(*********************************** G.D S.p.A. - Technical Department ***********************************
============= PROGRAM INFO ============
FOLDER:             TBD
MACHINES INVOLVED:  TBD 

============= DESCRIPTION =============
csp machine declaration

============= REVISIONS ===============
Date		Version	 	Author      	Description             
----------	-------		------------  	--------------------------------------------
2020/02/19 	0000.00	 	G.Imbriaco		

**********************************************************************************************************)
(*$R process_ref := prc; $*)
PROGRAM csp_case_glue_os_guns
VAR
	
	prc:											process;
	prc_path:										STRING;
	
END_VAR

VAR CONSTANT

END_VAR

_read_var_input();
_read_var_input();

_object_manager();

IF 	NOT objects_running()
THEN
	RETURN;	
END_IF

_read_process_image();

_mode_manager();

CASE process_get_mode(prc) of
	MODE_ABSENT,
	MODE_INACTIVE:
		RETURN;
	MODE_TEST:
		_handle_process_test();
END_CASE

_set_runtime_properties();

(********************************* BODY *********************************)

(************************************************************************)

_handle_messages();

_write_output();

ACTION _handle_messages:
;
END_ACTION

ACTION _handle_process_test:
;
END_ACTION

ACTION _mode_manager:
IF process_mode_req_is_pending(prc)
THEN
    process_apply_mode_req_first_step(prc);
    CASE process_get_mode(prc) OF
        MODE_TO_ABSENT:
			;
        MODE_TO_INACTIVE:
			;
        MODE_TO_TEST:
			;
        MODE_TO_OPERATIONAL:
			;
    END_CASE
    process_apply_mode_req_second_step(prc);
END_IF
END_ACTION

ACTION _object_manager:
IF objects_initialization()
THEN
	sub_process_init(
		object_name					:= 'csp_case_glue_os_guns.prc', 
		process						:= csp_case_glue_os.prc, 
		CONVERSION_this				:= prc);
		
	prc_path 						:= process_get_path(prc);
	
END_IF

IF objects_running()
THEN
	process_cycle(prc);

END_IF
END_ACTION

ACTION _read_process_image:
;
END_ACTION

ACTION _read_var_input:
;
END_ACTION

ACTION _set_runtime_properties:
;
END_ACTION

ACTION _write_output:
;
END_ACTION

END_PROGRAM

(* stored: Version 1.1.0.1, ProductVersion 3.1.4024.3
   POU csp_case_glue_os_guns: Id {7930b6d0-f08d-41ac-b582-de89390cbd0d}, SpecialFunc None
   Action _handle_messages: Id {87b0a46c-8804-4bf9-89e5-5c10ad04ebc5}
   Action _handle_process_test: Id {83e313a0-76a0-4627-9f63-acb10f0e0470}
   Action _mode_manager: Id {c8b35d26-52be-4fab-9e16-111ff99141cf}
   Action _object_manager: Id {25138427-b1c8-42f5-9446-12d02bda6cdd}
   Action _read_process_image: Id {fb82a24f-f56b-490f-b948-310cb91223d9}
   Action _read_var_input: Id {294d33f5-5264-4a69-91a8-4c6ec9a6eb38}
   Action _set_runtime_properties: Id {5c1795b7-654a-452a-a374-3ad46c73b8f9}
   Action _write_output: Id {c727ff96-0fee-416b-97e2-03cf1fe325b2} *)
